// TIA Portal V18 export
TYPE "DT_FML_REF"
// stored: IsFailsafeCompliant false
   STRUCT
      InData : Struct
         FHPP : Array[1..16] of Byte;
         FPC : Array[1..8] of Byte;
         FHPPplus : Array[1..10] of DInt;
      END_STRUCT;
      OutData : Struct
         FHPP : Array[1..16] of Byte;
         FPC : Array[1..8] of Byte;
         FHPPplus : Array[1..10] of DInt;
      END_STRUCT;
      Modbus : Bool;
      DeviceType : String[16];
      MemberID : Int;
      MemberIDmax : Int;
      Done : Bool;
      Err : Bool;
      PNU : Word;
      ActPNU : Word;
      ReqID : Int;
      RespID : Int;
      FPCC_Modus : Byte;
      FPCS_Modus : Byte;
      FPCC_Packet { S7_SetPoint := 'True'} : "DT_FML_PRM_FILE";
      FPCS_Packet { S7_SetPoint := 'True'} : "DT_FML_PRM_FILE";
      Subindex : Byte;
      ActSubindex : Byte;
      DatatypeWR : Byte;
      DatatypeRD : Byte;
      ParamValueWR : DInt;
      ParamValueRD : DInt;
   END_STRUCT;
END_TYPE
